TYPE CmpHMI :
STRUCT
	
	Title : STRING := '';
	Message : STRING := '';
	Timeout : TIME := T#0s;
	InformationOnly :BOOL;
	Trigger : BOOL;
	RespPositive : BOOL;
	RespNegative : BOOL;
	RespTimeout : BOOL;
	HeartbeatOK : BOOL;
	
END_STRUCT
END_TYPE

(* stored: Version 1.1.0.1, ProductVersion 3.1.4024.6
   DUT CmpHMI: Id {a3ef454c-ca33-4206-ba73-ebd402c6aace} *)
